// TIA Portal V19 export
FUNCTION "Assign Input" : Void   // FC4, LAD
{ S7_Optimized_Access := 'TRUE' }
// stored: SetENOAutomatically false
   VAR_INPUT
      Input1 : Bool;
      Input2 : Bool;
      Input3 : Bool;
      Input4 : Bool;
      Input5 : Bool;
      Input6 : Bool;
      Input7 : Bool;
      Input8 : Bool;
      Input9 : Bool;
      Input10 : Bool;
      Input11 : Bool;
      Input12 : Bool;
      Input13 : Bool;
      Input14 : Bool;
      InputSelection : Int;
   END_VAR
   VAR_OUTPUT
      Out : Bool;
      InputSelected : Int;
   END_VAR
BEGIN

REGION Network 1
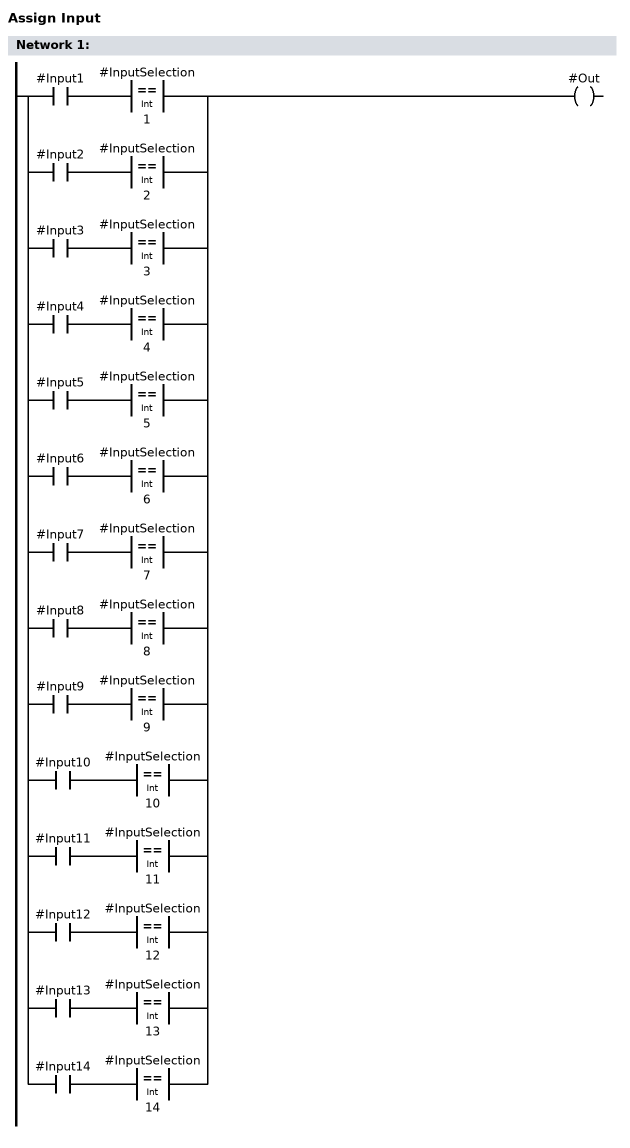
   RUNG wire#powerrail
      Contact( #Input1 )
      { S7_Templates := "SrcType := Int" } EQ_Contact(in1 := #InputSelection, in2 := 1)
      wire#w1
      Coil( #Out )
   END_RUNG
   RUNG wire#powerrail
      Contact( #Input2 )
      { S7_Templates := "SrcType := Int" } EQ_Contact(in1 := #InputSelection, in2 := 2)
   END_RUNG wire#w1
   RUNG wire#powerrail
      Contact( #Input3 )
      { S7_Templates := "SrcType := Int" } EQ_Contact(in1 := #InputSelection, in2 := 3)
   END_RUNG wire#w1
   RUNG wire#powerrail
      Contact( #Input4 )
      { S7_Templates := "SrcType := Int" } EQ_Contact(in1 := #InputSelection, in2 := 4)
   END_RUNG wire#w1
   RUNG wire#powerrail
      Contact( #Input5 )
      { S7_Templates := "SrcType := Int" } EQ_Contact(in1 := #InputSelection, in2 := 5)
   END_RUNG wire#w1
   RUNG wire#powerrail
      Contact( #Input6 )
      { S7_Templates := "SrcType := Int" } EQ_Contact(in1 := #InputSelection, in2 := 6)
   END_RUNG wire#w1
   RUNG wire#powerrail
      Contact( #Input7 )
      { S7_Templates := "SrcType := Int" } EQ_Contact(in1 := #InputSelection, in2 := 7)
   END_RUNG wire#w1
   RUNG wire#powerrail
      Contact( #Input8 )
      { S7_Templates := "SrcType := Int" } EQ_Contact(in1 := #InputSelection, in2 := 8)
   END_RUNG wire#w1
   RUNG wire#powerrail
      Contact( #Input9 )
      { S7_Templates := "SrcType := Int" } EQ_Contact(in1 := #InputSelection, in2 := 9)
   END_RUNG wire#w1
   RUNG wire#powerrail
      Contact( #Input10 )
      { S7_Templates := "SrcType := Int" } EQ_Contact(in1 := #InputSelection, in2 := 10)
   END_RUNG wire#w1
   RUNG wire#powerrail
      Contact( #Input11 )
      { S7_Templates := "SrcType := Int" } EQ_Contact(in1 := #InputSelection, in2 := 11)
   END_RUNG wire#w1
   RUNG wire#powerrail
      Contact( #Input12 )
      { S7_Templates := "SrcType := Int" } EQ_Contact(in1 := #InputSelection, in2 := 12)
   END_RUNG wire#w1
   RUNG wire#powerrail
      Contact( #Input13 )
      { S7_Templates := "SrcType := Int" } EQ_Contact(in1 := #InputSelection, in2 := 13)
   END_RUNG wire#w1
   RUNG wire#powerrail
      Contact( #Input14 )
      { S7_Templates := "SrcType := Int" } EQ_Contact(in1 := #InputSelection, in2 := 14)
   END_RUNG wire#w1
   // the same network as SCL:
   #Out := (#Input1 AND (#InputSelection = 1)) OR (#Input2 AND (#InputSelection = 2)) OR (#Input3 AND (#InputSelection = 3)) OR (#Input4 AND (#InputSelection = 4)) OR (#Input5 AND (#InputSelection = 5)) OR (#Input6 AND (#InputSelection = 6)) OR (#Input7 AND (#InputSelection = 7)) OR (#Input8 AND (#InputSelection = 8)) OR (#Input9 AND (#InputSelection = 9)) OR (#Input10 AND (#InputSelection = 10)) OR (#Input11 AND (#InputSelection = 11)) OR (#Input12 AND (#InputSelection = 12)) OR (#Input13 AND (#InputSelection = 13)) OR (#Input14 AND (#InputSelection = 14));
END_REGION
END_FUNCTION
